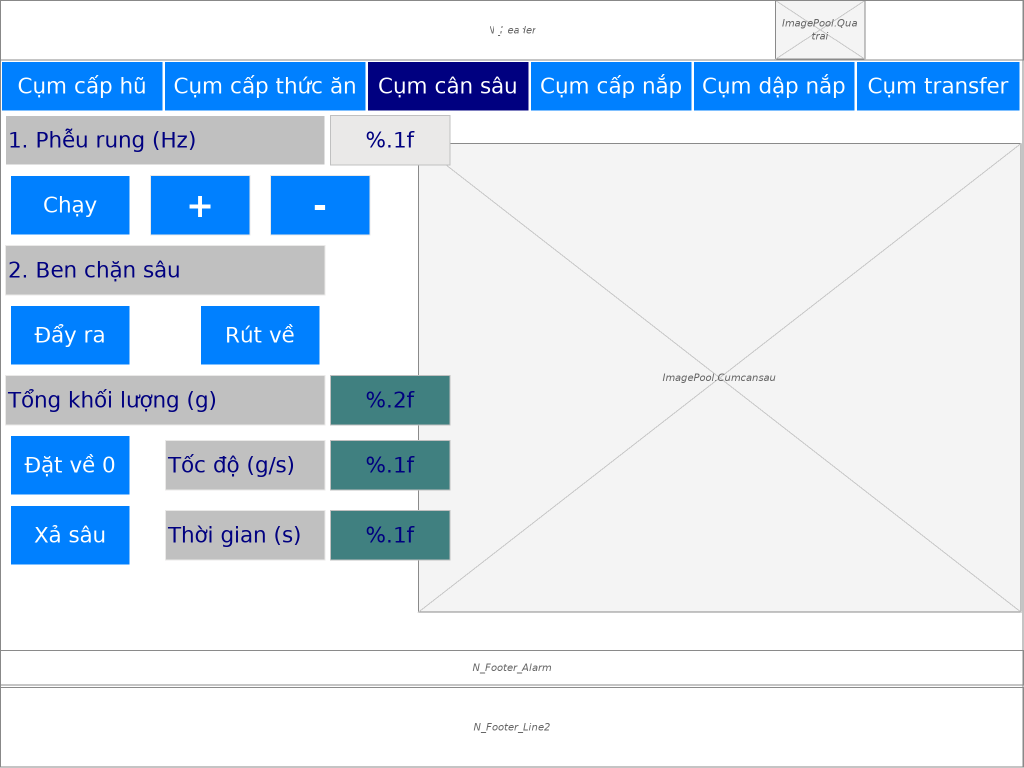
VISUALIZATION N_WormWeight2  // 1024x768
    Image (418,143 603x469), image: ImagePool.Cumcansau
    Rectangle (10,305 120x60), "Đẩy ra", colour toggle: PR_Line02.bCylinder_Block_Worm_Extend
        OnMouseDown: execute {
            PR_Line02.bCylinder_Block_Worm_Extend := TRUE;
            PR_Line02.bCylinder_Block_Worm_Retract := FALSE;
            PR_Line02.bxa := FALSE;
        }
    Rectangle (10,175 120x60), "Dừng", invisible if: not PR_Line02.bMotor_vibrating_funnel, input disabled if: not PR_Line02.bMotor_vibrating_funnel
        OnMouseDown: execute { PR_Line02.bMotor_vibrating_funnel := false; }
    Rectangle (200,305 120x60), "Rút về", colour toggle: PR_Line02.bCylinder_Block_Worm_Retract
        OnMouseDown: execute {
            PR_Line02.bCylinder_Block_Worm_Retract := TRUE;
            PR_Line02.bCylinder_Block_Worm_Extend := FALSE;
            PR_Line02.bxa := FALSE;
        }
    Frame (0,687 1024x80)
        shows N_Footer_Line2()
    Frame (0,0 1024x60)
        shows N_Header()
    Textfield (353,5 400x50), "MÀN HÌNH CHẠY TAY LINE 2"
    Rectangle (10,175 120x60), "Chạy", invisible if: PR_Line02.bMotor_vibrating_funnel, input disabled if: PR_Line02.bMotor_vibrating_funnel
        OnMouseDown: execute { PR_Line02.bMotor_vibrating_funnel := TRUE; PR_Line02.bxa := FALSE; }
    Rectangle (330,115 120x50), "%.1f", text variable: PR_Line02.fb_WormWeight.fSpeed_vibrating_funnel_Manual
        OnMouseDown: write PR_Line02.fb_WormWeight.fSpeed_vibrating_funnel_Manual via VisuDialogs.Numpad
        OnMouseDown: execute { PR_Line02.bxa := FALSE; }
    Rectangle (150,175 100x60), "+", colour toggle: PR_Line02.bUp_vibrating_funnel
        OnMouseDown: execute { PR_Line02.bUp_vibrating_funnel := TRUE; PR_Line02.bxa := FALSE; }
    Rectangle (270,175 100x60), "-", colour toggle: PR_Line02.bDown_vibrating_funnel
        OnMouseDown: execute { PR_Line02.bDown_vibrating_funnel := TRUE; PR_Line02.bxa := FALSE; }
    Rectangle (330,375 120x50), "%.2f", text variable: PR_Line02.fb_WormWeight.fWeight_Worm
    Rectangle (10,435 120x60), "Đặt về 0"
        tap PR_Line02.bZero_Loadcell_Worm
        OnMouseDown: execute { PR_Line02.bxa := FALSE; }
        OnMouseUp: execute { PR_Line02.bZero_Loadcell_Worm := TRUE; }
    Rectangle (330,440 120x50), "%.1f", text variable: PR_Line02.fb_WormWeight.fFlow_Worm
    Image (775,0 90x59), input disabled if: bResetAuto1, image: ImagePool.Qua trai
        OnMouseClick: change screen: N_WormWeight1
        OnMouseClick: execute { MAIN.bModeManual := TRUE; MAIN.bModeAuto := FALSE; }
    Rectangle (1,61 162x50), "Cụm cấp hũ"
        OnMouseClick: change screen: N_JarSupply2
    Rectangle (164,61 202x50), "Cụm cấp thức ăn"
        OnMouseClick: change screen: N_FoodSupply2
    Rectangle (367,61 162x50), "Cụm cân sâu"
        OnMouseClick: change screen: N_WormWeight2
    Rectangle (530,61 162x50), "Cụm cấp nắp"
        OnMouseClick: change screen: N_LidSupply2
    Rectangle (693,61 162x50), "Cụm dập nắp"
        OnMouseClick: change screen: N_LidPressing2
    Rectangle (856,61 164x50), "Cụm transfer"
        OnMouseClick: change screen: N_Tranfer2
    Rectangle (5,375 320x50), "Tổng khối lượng (g)"
    Rectangle (5,115 320x50), "1. Phễu rung (Hz)"
    Rectangle (5,245 320x50), "2. Ben chặn sâu"
    Rectangle (165,440 160x50), "Tốc độ (g/s)"
    Rectangle (165,510 160x50), "Thời gian (s)"
    Rectangle (10,505 120x60), "Xả sâu", colour toggle: PR_Line02.xasau
        OnMouseDown: execute { PR_Line02.xasau := TRUE; PR_Line02.bxa := true; }
    Rectangle (330,510 120x50), "%.1f", text variable: PR_Line02.fb_WormWeight.fTime
    Frame (0,650 1024x35)
        shows N_Footer_Alarm()
END_VISUALIZATION

(* stored: Version 1.1.0.1, ProductVersion 3.1.4024.12
   Visu N_WormWeight2: Id {1d1b582c-3b9e-49d8-964c-79fe2870856f} *)
